// TIA Portal project "Programma PLC smistamento pacchi colore" (V15.1)
// Vorlageprojekt für das Buch mit Zielsystem S7-1200

(* hardware
DEVICE "S7-1200-Station_1"  S7-1200 Station
   slot 0: "Baugruppenträger_0"  Rack  V1.0
   slot 1: "PLC_1"  CPU 1211C DC/DC/DC  6ES7 211-1AE40-0XB0  V4.1
*)

// ===== PLC "PLC_1"  CPU 1211C DC/DC/DC =====

VAR_GLOBAL   // PLC tag table "Standard-Variablentabelle"
   "Tag_1" AT %A0.0 : Bool;
   "Tag_2" AT %E0.0 : Bool;
   "Tag_3" AT %E0.1 : Bool;
   "Motore_blu" AT %Q0.1 : Bool;
   "Motore_verde" AT %Q0.2 : Bool;
   "Sensore_presenza_pacchi" AT %I0.2 : Bool;
   "Sensore_colore_pacchi" AT %I0.3 : Bool;
   "Motore_rulli" AT %Q0.3 : Bool;
   "Rulli_Destra" AT %Q0.4 : Bool;
   "Rulli_Sinistra" AT %Q0.5 : Bool;
   "Sensore_presenza_pacco_blu" AT %I0.4 : Bool;
   "Sensore_presenza_pacco_verde" AT %I0.5 : Bool;
   "Pacchi verdi rimanenti" AT %MB0 : USInt;
   "Pacchi blu rimanenti" AT %MB1 : USInt;
   "Stato Sensore presenza pacchi" AT %M2.0 : Bool;
   "Stato Sensore pacco blu" AT %M2.1 : Bool;
   "Stato Sensore pacco verde" AT %M2.2 : Bool;
   "Loop" AT %M2.3 : Bool;
   "Pulsante Start" AT %I0.6 : Bool;
   "Pulsante Pausa" AT %I0.7 : Bool;
   "Numero Pacchi Blu" AT %QD30 : DInt;
   "Numero Pacchi Verdi" AT %QD34 : DInt;
   "Motore nastro principale" AT %Q0.6 : Bool;
   "Emettitore pacchi" AT %Q0.7 : Bool;
   "Luce pulsante start" AT %Q1.0 : Bool;
   "Luce pulsante stop" AT %Q1.1 : Bool;
END_VAR

DATA_BLOCK "Motori"   // DB1
{ S7_Optimized_Access := 'TRUE' }
VERSION : 0.1
   VAR
      "Stato Motore N_Blu" : Bool;   // Variabile di stato del nastro dei pacchi blu
      "Stato Motore N_Verde" : Bool;   // Variabile di stato del nastro dei pacchi verdi
      "Stato Motore Rulli" : Bool;   // Variavile di stato per l'azionamento dei rulli
      "Direzione Rulli" : Bool;   // Variabile che indica la direzione dei rulli (0=destra; 1= sinistra)
   END_VAR
BEGIN
END_DATA_BLOCK

FUNCTION "Azionamento Motori" : Void   // FC1, LAD
{ S7_Optimized_Access := 'TRUE' }
VERSION : 0.1
   VAR_INPUT
      "Presenza Pacco" : Bool;   // Sensore per vedere se c'è un pacco
      "Colore pacco" : Bool;   // (0=verde; 1=blu)
      "Sensore pacco blu" : Bool;   // Sensore presenza pacco blu sul nastro
      "Sensore pacco verde" : Bool;   // Sensore presenza pacco verde sul nastro
   END_VAR
   VAR_OUTPUT
      "Motore Rulli" : Bool;   // Motore rulli che direzionano il pacco
      Destra : Bool;   // Comando per direzionare a destra
      Sinistra : Bool;   // Comando per direzionare a sinistra
      "Motore Nastro Blu" : Bool;   // Motore nastro trasportatore pacchi blu
      "Motore Nastro Verde" : Bool;   // Motore nastro trasportatore pacchi verdi
   END_VAR
   VAR_TEMP   // added for the SCL form of the ladder/FBD networks
      _w1 : Bool;
   END_VAR
BEGIN

REGION Network 1: Variavile di stato per l'azionamento dei rulli
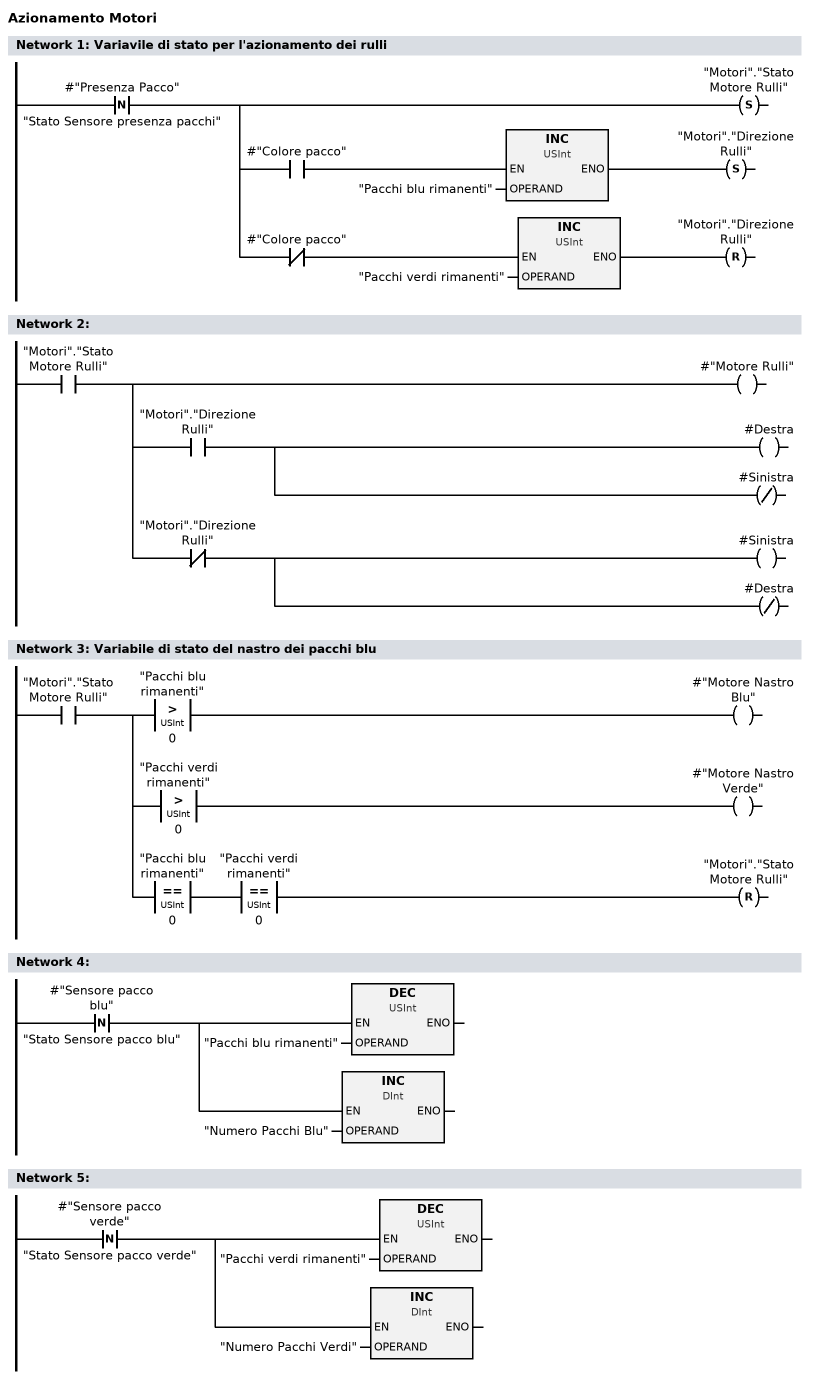
   RUNG wire#powerrail
      N_Contact(operand := #"Presenza Pacco", bit := "Stato Sensore presenza pacchi")
      wire#w1
      S_Coil( "Motori"."Stato Motore Rulli" )
   END_RUNG
   RUNG wire#w1
      Contact( #"Colore pacco" )
      { S7_Templates := "DestType := USInt" } Inc( "Pacchi blu rimanenti" )
      S_Coil( "Motori"."Direzione Rulli" )
   END_RUNG
   RUNG wire#w1
      I_Contact( #"Colore pacco" )
      { S7_Templates := "DestType := USInt" } Inc( "Pacchi verdi rimanenti" )
      R_Coil( "Motori"."Direzione Rulli" )
   END_RUNG
   // the same network as SCL:
   #_w1 := NOT #"Presenza Pacco" AND "Stato Sensore presenza pacchi";   // falling edge of #"Presenza Pacco"
   "Stato Sensore presenza pacchi" := #"Presenza Pacco";
   IF #_w1 THEN "Motori"."Stato Motore Rulli" := TRUE; END_IF;
   IF #_w1 AND #"Colore pacco" THEN
       "Pacchi blu rimanenti" := "Pacchi blu rimanenti" + 1;
       "Motori"."Direzione Rulli" := TRUE;
   END_IF;
   IF #_w1 AND NOT #"Colore pacco" THEN
       "Pacchi verdi rimanenti" := "Pacchi verdi rimanenti" + 1;
       "Motori"."Direzione Rulli" := FALSE;
   END_IF;
END_REGION

REGION Network 2
   RUNG wire#powerrail
      Contact( "Motori"."Stato Motore Rulli" )
      wire#w1
      Coil( #"Motore Rulli" )
   END_RUNG
   RUNG wire#w1
      Contact( "Motori"."Direzione Rulli" )
      wire#w2
      Coil( #Destra )
   END_RUNG
   RUNG wire#w2
      I_Coil( #Sinistra )
   END_RUNG
   RUNG wire#w1
      I_Contact( "Motori"."Direzione Rulli" )
      wire#w3
      Coil( #Sinistra )
   END_RUNG
   RUNG wire#w3
      I_Coil( #Destra )
   END_RUNG
   // the same network as SCL:
   #"Motore Rulli" := "Motori"."Stato Motore Rulli";
   #Destra := "Motori"."Stato Motore Rulli" AND "Motori"."Direzione Rulli";
   #Sinistra := NOT #Destra;
   #Sinistra := "Motori"."Stato Motore Rulli" AND NOT "Motori"."Direzione Rulli";
   #Destra := NOT #Sinistra;
END_REGION

REGION Network 3: Variabile di stato del nastro dei pacchi blu
   RUNG wire#powerrail
      Contact( "Motori"."Stato Motore Rulli" )
      wire#w1
      { S7_Templates := "SrcType := USInt" } GT_Contact(in1 := "Pacchi blu rimanenti", in2 := 0)
      Coil( #"Motore Nastro Blu" )
   END_RUNG
   RUNG wire#w1
      { S7_Templates := "SrcType := USInt" } GT_Contact(in1 := "Pacchi verdi rimanenti", in2 := 0)
      Coil( #"Motore Nastro Verde" )
   END_RUNG
   RUNG wire#w1
      { S7_Templates := "SrcType := USInt" } EQ_Contact(in1 := "Pacchi blu rimanenti", in2 := 0)
      { S7_Templates := "SrcType := USInt" } EQ_Contact(in1 := "Pacchi verdi rimanenti", in2 := 0)
      R_Coil( "Motori"."Stato Motore Rulli" )
   END_RUNG
   // the same network as SCL:
   #"Motore Nastro Blu" := "Motori"."Stato Motore Rulli" AND ("Pacchi blu rimanenti" > 0);
   #"Motore Nastro Verde" := "Motori"."Stato Motore Rulli" AND ("Pacchi verdi rimanenti" > 0);
   IF "Motori"."Stato Motore Rulli" AND ("Pacchi blu rimanenti" = 0) AND ("Pacchi verdi rimanenti" = 0) THEN
       "Motori"."Stato Motore Rulli" := FALSE;
   END_IF;
END_REGION

REGION Network 4
   RUNG wire#powerrail
      N_Contact(operand := #"Sensore pacco blu", bit := "Stato Sensore pacco blu")
      wire#w1
      { S7_Templates := "DestType := USInt" } Dec( "Pacchi blu rimanenti" )
   END_RUNG
   RUNG wire#w1
      { S7_Templates := "DestType := DInt" } Inc( "Numero Pacchi Blu" )
   END_RUNG
   // the same network as SCL:
   #_w1 := NOT #"Sensore pacco blu" AND "Stato Sensore pacco blu";   // falling edge of #"Sensore pacco blu"
   "Stato Sensore pacco blu" := #"Sensore pacco blu";
   IF #_w1 THEN
       "Pacchi blu rimanenti" := "Pacchi blu rimanenti" - 1;
       "Numero Pacchi Blu" := "Numero Pacchi Blu" + 1;
   END_IF;
END_REGION

REGION Network 5
   RUNG wire#powerrail
      N_Contact(operand := #"Sensore pacco verde", bit := "Stato Sensore pacco verde")
      wire#w1
      { S7_Templates := "DestType := USInt" } Dec( "Pacchi verdi rimanenti" )
   END_RUNG
   RUNG wire#w1
      { S7_Templates := "DestType := DInt" } Inc( "Numero Pacchi Verdi" )
   END_RUNG
   // the same network as SCL:
   #_w1 := NOT #"Sensore pacco verde" AND "Stato Sensore pacco verde";   // falling edge of #"Sensore pacco verde"
   "Stato Sensore pacco verde" := #"Sensore pacco verde";
   IF #_w1 THEN
       "Pacchi verdi rimanenti" := "Pacchi verdi rimanenti" - 1;
       "Numero Pacchi Verdi" := "Numero Pacchi Verdi" + 1;
   END_IF;
END_REGION
END_FUNCTION

FUNCTION "MHJ-PLC-Lab-Function-S71200" : Void   // FC9000, SCL
{ S7_Optimized_Access := 'TRUE' }
VERSION : 0.1
   VAR_TEMP
      rdTimeReturn : Int;
      outputTime : DTL;
      SyncVal : Byte;
      forVal : Int;
      forVal_2 : Int;
      Value : Byte;
   END_VAR
   VAR CONSTANT
      CompVal : Byte := 16#34;
      Value_01 : Byte := 16#11;
      Value_01_DW : DWord := 16#A165_D992;
      Value_02_DW : DWord := 16#58BE_4401;
   END_VAR
BEGIN

   #Value:=PEEK(area := 16#82,
        dbNumber := 0,
        byteOffset := 511);
   #Value := #Value + 1;

   POKE(area := 16#82,
        dbNumber := 0,
        byteOffset := 511,
        value := #Value);

   POKE(area:=16#81,
        dbNumber:=0,
        byteOffset:=1016,
        value:=#Value_01_DW);
   POKE(area := 16#81,
        dbNumber := 0,
        byteOffset := 1020,
        value := #Value_02_DW);

   POKE(area := 16#81,
        dbNumber := 0,
        byteOffset := 511,
        value := B#16#00);

   FOR #forVal := 0 TO 120 DO
       FOR #forVal_2:=0 TO 10 DO
           #rdTimeReturn:=RD_SYS_T(#outputTime);
           #rdTimeReturn := WR_SYS_T(#outputTime);
           #rdTimeReturn := RD_SYS_T(#outputTime);
           #rdTimeReturn := WR_SYS_T(#outputTime);
       END_FOR;
       #SyncVal:= PEEK(area := 16#81,
                      dbNumber := 0,
                      byteOffset := 511);
       IF #SyncVal = #CompVal THEN
          GOTO M_1;
       END_IF;
   END_FOR;
   RETURN;

   M_1:
   POKE(area := 16#81,
        dbNumber := 0,
        byteOffset := 511,
        value := B#16#0);
END_FUNCTION

ORGANIZATION_BLOCK "Main"   // OB1, LAD, ProgramCycle
TITLE = "Main Program Sweep (Cycle)"
{ S7_Optimized_Access := 'TRUE' }
VERSION : 0.1
   VAR_INPUT
      Initial_Call : Bool;   // Initial call of this OB
      Remanence : Bool;   // =True, if remanent data are available
   END_VAR
BEGIN

REGION Network 1: Konnektierungsbaustein für PLC-Lab
   // Im Netzwerk 1 wird der Konnektierungsbaustein für PLC-Lab aufgerufen.
   // Dieser Aufruf darf nicht entfernt werden!
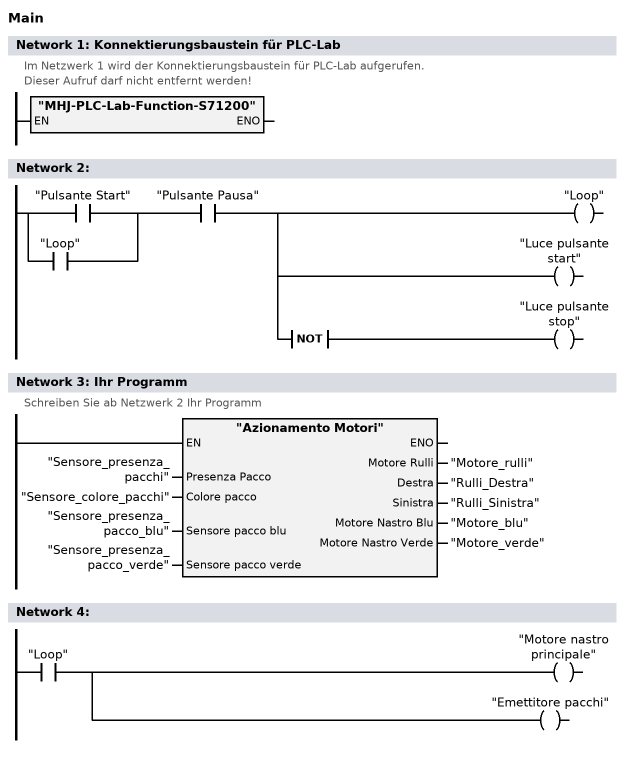
   RUNG wire#powerrail
      "MHJ-PLC-Lab-Function-S71200"()
   END_RUNG
   // the same network as SCL:
   "MHJ-PLC-Lab-Function-S71200"();
END_REGION

REGION Network 2
   RUNG wire#powerrail
      Contact( "Pulsante Start" )
      wire#w1
      Contact( "Pulsante Pausa" )
      wire#w2
      Coil( "Loop" )
   END_RUNG
   RUNG wire#powerrail
      Contact( "Loop" )
   END_RUNG wire#w1
   RUNG wire#w2
      Coil( "Luce pulsante start" )
   END_RUNG
   RUNG wire#w2
      Not()
      Coil( "Luce pulsante stop" )
   END_RUNG
   // the same network as SCL:
   "Loop" := ("Pulsante Start" OR "Loop") AND "Pulsante Pausa";
   "Luce pulsante start" := "Loop";
   "Luce pulsante stop" := NOT "Loop";
END_REGION

REGION Network 3: Ihr Programm
   // Schreiben Sie ab Netzwerk 2 Ihr Programm
   RUNG wire#powerrail
      "Azionamento Motori"("Presenza Pacco" := "Sensore_presenza_pacchi", "Colore pacco" := "Sensore_colore_pacchi", "Sensore pacco blu" := "Sensore_presenza_pacco_blu", "Sensore pacco verde" := "Sensore_presenza_pacco_verde", "Motore Rulli" => "Motore_rulli", Destra => "Rulli_Destra", Sinistra => "Rulli_Sinistra", "Motore Nastro Blu" => "Motore_blu", "Motore Nastro Verde" => "Motore_verde")
   END_RUNG
   // the same network as SCL:
   "Azionamento Motori"("Presenza Pacco" := "Sensore_presenza_pacchi",
                        "Colore pacco" := "Sensore_colore_pacchi",
                        "Sensore pacco blu" := "Sensore_presenza_pacco_blu",
                        "Sensore pacco verde" := "Sensore_presenza_pacco_verde",
                        "Motore Rulli" => "Motore_rulli",
                        Destra => "Rulli_Destra",
                        Sinistra => "Rulli_Sinistra",
                        "Motore Nastro Blu" => "Motore_blu",
                        "Motore Nastro Verde" => "Motore_verde");
END_REGION

REGION Network 4
   RUNG wire#powerrail
      Contact( "Loop" )
      wire#w1
      Coil( "Motore nastro principale" )
   END_RUNG
   RUNG wire#w1
      Coil( "Emettitore pacchi" )
   END_RUNG
   // the same network as SCL:
   "Motore nastro principale" := "Loop";
   "Emettitore pacchi" := "Loop";
END_REGION
END_ORGANIZATION_BLOCK